FUNCTION atan2Fun : lreal
VAR_INPUT
	y:LREAL;
	x:LREAL;
END_VAR
VAR
END_VAR

//atan2(y,x)
IF ABS(x)<=0.0000001 THEN
	IF y>0 THEN
		atan2Fun:=pi/2;
	ELSE
		atan2Fun:=-pi/2;
	END_IF
ELSE
	IF x>0 THEN
		atan2Fun:=ATAN(y/x);
	ELSE
		IF y<0 THEN
			atan2Fun:=ATAN(y/x)-pi;	
		ELSE
			atan2Fun:=ATAN(y/x)+pi;
		END_IF
	END_IF
END_IF

END_FUNCTION

(* stored: Version 1.1.0.1, ProductVersion 3.1.4024.2
   POU atan2Fun: Id {352f4838-6b04-4472-b751-8203570ca69c}, SpecialFunc None *)
